FUNCTION_BLOCK SUBSCRIBE_1 (* Single-variable Subscriber *)
  (* Standard: 61499-1-3.2 *)
  (* Version 0.2, 2008-06-04, JHC, Holobloc Inc, Updated DOCTYPE. *)
  (* Version 0.1, 2001-04-24, JHC, Rockwell Automation, XML version *)
  (* Version 0.0, 1998-12-01, JHC, Rockwell Automation, SRC version *)
  (* Compiler header: package fb.rt.net; *)
  (* Compiler Java IBM VisualAge 3.0 *)
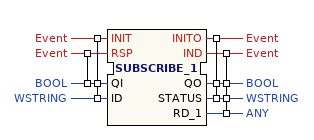
  EVENT_INPUT
    INIT WITH QI, ID; (* Service Initialization *)
    RSP WITH QI; (* Service Response *)
  END_EVENT
  EVENT_OUTPUT
    INITO WITH QO, STATUS; (* Initialization Confirm *)
    IND WITH QO, STATUS, RD_1; (* Service Indication *)
  END_EVENT
  VAR_INPUT
    QI : BOOL; (* Event Input Qualifier *)
    ID : WSTRING; (* Connection Identifier *)
  END_VAR
  VAR_OUTPUT
    QO : BOOL; (* Event Output Qualifier *)
    STATUS : WSTRING; (* Service Status *)
    RD_1 : ANY; (* Subscribed Data *)
  END_VAR
END_FUNCTION_BLOCK
